(* IEC 61131-3 sources: repolevel_ST_code_completion/dataset/generation_context_ground_truth/PID_controller, 4 files *)

(* ---- HeatExchanger.st ---- *)
VAR
	now: TIME;
	lastTime: TIME;
	lastPV:REAL := 140;
	A: REAL;
	B: REAL;
	delta_t: REAL;
END_VAR
VAR CONSTANT
	millis: REAL := 1000;
END_VAR

now := TIME();
IF ((now - lastTime) > Sample_time) THEN
	delta_t := TIME_TO_REAL(Sample_time)/millis;
	A := EXP(-delta_t/Tp);
	B := 1 - A;
	C := 2;

	//PV := A * lastPV + B * Kp * CO + C;
	PV := 0.987 * lastPV - 0.00679 * CO + C;
	lastPV := PV;

	lastTime := now;
END_IF

(* ---- HeatExchanger2.st ---- *)
VAR
	now: TIME;
	lastTime: TIME := T#0s;
	delta_t: REAL;
	heat_flow: REAL;
	lastTemp: REAL;
END_VAR
VAR CONSTANT
	millis: REAL := 1000;
END_VAR

now := TIME();
IF ((now - lastTime) > Sample_time) THEN
	delta_t := TIME_TO_REAL(Sample_time)/millis;

	//First calculate net heat
	//Heat_In is our heat source
	//Second term is heat flow depending on temperature difference
	//Obs: At start, set lastTime to start temp Temp_In
	IF lastTime = T#0S THEN
		lastTemp := Temp_In;
	END_IF
	heat_flow := Heat_In - U * (lastTemp - Temp_Out);

	//Second: calculate temperature change due to heat_flow
	Temp := lastTemp + heat_flow * delta_t / TC;

	//Update variables for next iteration
	lastTemp := Temp;
	lastTime := now;
END_IF;

(* ---- PID_controller.st ---- *)
VAR CONSTANT
	millis: UINT := 1000;
END_VAR
VAR
	now: TIME := T#0S;
	lastTime: TIME := T#0S;
	err: REAL := 0; //Process error
	lastCO_P: REAL := 0;  //Used for calculation of the derivative term
	delta_t: REAL;
	lastPV: REAL := 0;
END_VAR

//Check parameters
//Ti division by zero
IF Ti = 0 THEN
	Ti := 1;
END_IF

//Update PID parameters every sampleTime
now := TIME();
IF ((now - lastTime) > SampleTime) THEN
	err := SP - PV;
	delta_t := TIME_TO_REAL(SampleTime)/millis;
	CO_P := Kc * err;
	CO_I := CO_I + 1/Ti * CO_P * delta_t;
	//Add wind-up for CO_I
	IF CO_I < LowerLimit THEN
		CO_I := LowerLimit;
	ELSIF CO_I > UpperLimit THEN
		CO_I := UpperLimit;
	END_IF;

	//Observe that d(err)/dt = d(SP)/dt - d(PV)/dt
	//If SP constant,
	//d(err)/dt = - d(PV)/dt
	//Good: no output spikes
	//Bad: some processes need more aggressive tuning
	IF delta_t <> 0 THEN
		CO_D := Td * (PV - lastPV)/delta_t;
	END_IF;

	//A different approch would be with a tunable filter

	CO := CO_P + CO_I + CO_D;
	//Add wind-up for CO
	IF CO < LowerLimit THEN
		CO := LowerLimit;
	ELSIF CO > UpperLimit THEN
		CO := UpperLimit;
	END_IF;

	lastTime := now;
	lastPV := PV;
END_IF;

(* ---- Tank.st ---- *)
VAR
	now: TIME;
	lastTime: TIME;
	proc_sum_in: REAL := 0;
	proc_sum_out: REAL := 0;
	temp: REAL;
	millis: UINT := 1000;
	proc_out: REAL;
END_VAR

now := TIME();
IF ((now - lastTime) > SampleTime) THEN
	Level := Level +  TIME_TO_REAL(SampleTime)/millis * (Process_In - Process_Out);
	IF Level < Lower_limit THEN
		Level := Lower_limit;
	ELSIF Level > Upper_limit THEN
		Level := Upper_limit;
	END_IF;
	lastTime := now;
END_IF;
